// TIA Portal V16 export
// export: Created 2021-07-03T20:57:07.0651865Z, ExportSetting WithDefaults, DisplayName Totally Integrated Automation Portal, DisplayVersion V16, DisplayName TIA Portal Version Control Interface, DisplayVersion V16, DisplayName TIA Portal Openness, DisplayVersion V16, DisplayName STEP 7 Professional, DisplayVersion V16, DisplayName STEP 7 Safety, DisplayVersion V16, DisplayName WinCC Professional, DisplayVersion V16
FUNCTION "ISO_on_TCP-Blank" : Void   // FC2, FBD
{ S7_Optimized_Access := 'TRUE' }
VERSION : 0.1
// stored: AutoNumber false, IsIECCheckEnabled false, SetENOAutomatically false, UDAEnableTagReadback false
BEGIN

REGION Network 1
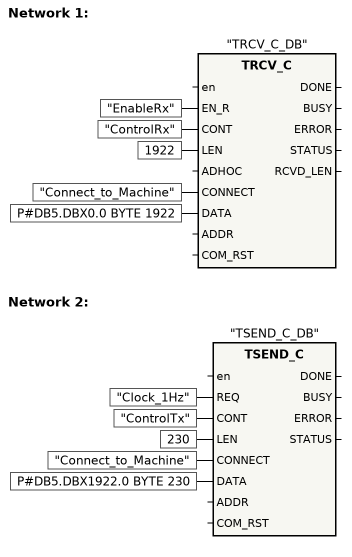
   "TRCV_C_DB"(EN_R := "EnableRx",   // TRCV_C
               CONT := "ControlRx",
               LEN := 1922,
               CONNECT := "Connect_to_Machine",
               DATA := P#DB5.DBX0.0 BYTE 1922);
END_REGION

REGION Network 2
   "TSEND_C_DB"(REQ := "Clock_1Hz",   // TSEND_C
                CONT := "ControlTx",
                LEN := 230,
                CONNECT := "Connect_to_Machine",
                DATA := P#DB5.DBX1922.0 BYTE 230);
END_REGION

REGION Network 3: Heartbeat
   // add the heartbeat here.
END_REGION
END_FUNCTION
